// TIA Portal V17 export
// export: Created 2025-05-22T05:59:34.6834771Z, ExportSetting WithDefaults, DisplayName Totally Integrated Automation Portal, DisplayVersion V17 Update 8, DisplayName TIA Portal Openness, DisplayVersion V17 Update 8, DisplayName TIA Portal Version Control Interface, DisplayVersion V17, DisplayName SINAMICS Startdrive Advanced, DisplayVersion V17 SP2, DisplayName SINAMICS Startdrive G110M, G120, G120C, G120D, G120P, G115D, DisplayVersion V17 SP2, DisplayName SINAMICS Startdrive G130, G150, S120, S150, SINAMICS MV, S210, DisplayVersion V17 SP2, DisplayName STEP 7 Professional, DisplayVersion V17 Update 8, DisplayName SINUMERIK ONE STEP 7 Toolbox, DisplayVersion V17 Update 12, DisplayName SINUMERIK ONE PLC Basic Program Plus, DisplayVersion V17 Update 12, DisplayName SINUMERIK 840D sl STEP 7 Toolbox, DisplayVersion V17 Update 12, DisplayName STEP 7 Safety, DisplayVersion V17 Update 6, DisplayName WinCC Advanced, DisplayVersion V17 Update 8
FUNCTION_BLOCK "FB10200_PYROMETERS"   // FB10200, LAD
{ S7_Optimized_Access := 'FALSE' }
AUTHOR : ETXETAR
VERSION : 1.0
// stored: AutoNumber false, IsIECCheckEnabled false, SetENOAutomatically false, UDAEnableTagReadback false
   VAR_INPUT
      OPTIONS_0 : Byte := 2#0000_0000;   // OPTIONS 0
      DEVICE_STATUS_SENSOR_INPUT : Real;   // DEVICE STATUS SENSOR INPUT
      PROCESS_TEMP_SENSOR_INPUT : Real;   // PROCESS TEMPERATURE SENSOR INPUT
      HEAD_TEMP_SENSOR_INPUT : Real;   // HEAD TEMPERATURE SENSOR INPUT
      T1_TEMP_SENSOR_INPUT : Real;   // T1 TEMPERATURE SENSOR INPUT
      T2_TEMP_SENSOR_INPUT : Real;   // T2 TEMPERATURE SENSOR INPUT
      CURRENT_EMISSIVITY_SENSOR_INPUT : Real;   // CURRENT EMISSIVITY SENSOR INPUT
      CURRENT_TRANSMISSION_SENSOR_INPUT : Real;   // CURRENT TRANSMISSION SENSOR INPUT
      STATION_CYCLE_RUNNING : Bool;   // SATION CYCLE RUNNING
   END_VAR
   VAR_OUTPUT
      PROCESS_TEMP_LOW_WARNING : Bool;   // PROCESS TEMPERATURE LOW WARNING
      PROCESS_TEMP_HIGH_WARNING : Bool;   // PROCESS TEMPERATURE HIGH WARNING
      HEAD_TEMP_LOW_WARNING : Bool;   // HEAD TEMPERATURE LOW WARNING
      HEAD_TEMP_HIGH_WARNING : Bool;   // HEAD TEMPERATURE HIGH WARNING
      EMISSIVITY_LOW_WARNING : Bool;   // EMISSIVITY LOW WARNING
      EMISSIVITY_HIGH_WARNING : Bool;   // EMISSIVITY HIGH WARNING
      PROCESS_TEMP_LOW_ALARM : Bool;   // PROCESS TEMPERATURE LOW ALARM
      PROCESS_TEMP_HIGH_ALARM : Bool;   // PROCESS TEMPERATURE HIGH ALARM
      HEAD_TEMP_LOW_ALARM : Bool;   // HEAD TEMPERATURE LOW ALARM
      HEAD_TEMP_HIGH_ALARM : Bool;   // HEAD TEMPERATURE HIGH ALARM
      EMISSIVITY_LOW_ALARM : Bool;   // EMISSIVITY LOW ALARM
      EMISSIVITY_HIGH_ALARM : Bool;   // EMISSIVITY HIGH ALARM
   END_VAR
   VAR DB_SPECIFIC
      ANY_ACTIVE_ALARM : Bool;   // ANY ACTIVE ALARM
      SEOC_ALARMS : Bool;   // STOP END OF CYCLE ALARMS
      RHP_SEOC_ALARMS : Bool;   // RETURN HOME POSITION AND STOP END OF CYCLE ALARMS
      IS_SEOC_ALARMS : Bool;   // INMEDIATE STOP AND STOP END OF CYCLE ALARMS
      UNIT_NUMBER : Int;   // UNIT NUMBER
      PROCESS_TEMP_SETTINGS : Struct
         LOW_WARNING_VALUE : Real;   // LOW WARNING VALUE
         HIGH_WARNING_VALUE : Real;   // HIGH WARNING VALUE
         LOW_ALARM_VALUE : Real;   // LOW ALARM VALUE
         HIGH_ALARM_VALUE : Real;   // HIGH ALARM VALUE
      END_STRUCT;
      HEAD_TEMP_SETTINGS : Struct
         LOW_WARNING_VALUE : Real;   // LOW WARNING VALUE
         HIGH_WARNING_VALUE : Real;   // HIGH WARNING VALUE
         LOW_ALARM_VALUE : Real;   // LOW ALARM VALUE
         HIGH_ALARM_VALUE : Real;   // HIGH ALARM VALUE
      END_STRUCT;
      EMISSIVITY_SETTINGS : Struct
         LOW_WARNING_VALUE : Real;   // LOW WARNING VALUE
         HIGH_WARNING_VALUE : Real;   // HIGH WARNING VALUE
         LOW_ALARM_VALUE : Real;   // LOW ALARM VALUE
         HIGH_ALARM_VALUE : Real;   // HIGH ALARM VALUE
      END_STRUCT;
      TIMERS : Struct
         PROCESS_TEMP_LOW_ALARM_TIMER : TON_TIME;
         PROCESS_TEMP_LOW_WARNING_TIMER : TON_TIME;
         PROCESS_TEMP_HIGH_ALARM_TIMER : TON_TIME;
         PROCESS_TEMP_HIGH_WARNING_TIMER : TON_TIME;
         HEAD_TEMP_LOW_ALARM_TIMER : TON_TIME;
         HEAD_TEMP_LOW_WARNING_TIMER : TON_TIME;
         HEAD_TEMP_HIGH_ALARM_TIMER : TON_TIME;
         HEAD_TEMP_HIGH_WARNING_TIMER : TON_TIME;
         EMISSIVITY_LOW_ALARM_TIMER : TON_TIME;
         EMISSIVITY_LOW_WARNING_TIMER : TON_TIME;
         EMISSIVITY_HIGH_ALARM_TIMER : TON_TIME;
         EMISSIVITY_HIGH_WARNING_TIMER : TON_TIME;
      END_STRUCT;
   END_VAR
   VAR_TEMP
      INPUTS_MASK : Byte;   // INPUT MASK
      O_BYTE_0 : Struct   // OPTIONS BYTE 0
         PROCESS_TEMP_WRNS_ENABLED : Bool;   // PROCESS TEMPERATURE WARNINGS ENABLED
         PROCESS_TEMP_ALARMS_ENABLED : Bool;   // PROCESS TEMPERATURE ALARMS ENABLED
         HEAD_TEMP_WRNS_ENABLED : Bool;   // HEAD TEMPERATURE WARNINGS ENABLED
         HEAD_TEMP_ALARMS_ENABLED : Bool;   // HEAD TEMPERATURE ALARMS ENABLED
         EMISSIVITY_WRNS_ENABLED : Bool;   // EMISSIVITY WARNINGS ENABLED
         EMISSIVITY_ALARMS_ENABLED : Bool;   // EMISSIVITY ALARMS ENABLED
         SPARE_6 : Bool;   // SPARE
         SPARE_7 : Bool;   // SPARE
      END_STRUCT;
      DB_NUMBER : DInt;   // DB NUMBER FOR ALARM AND HELP DECODING
   END_VAR
   VAR_TEMP   // added for the SCL form of the ladder/FBD networks
      _w1 : Bool;
   END_VAR
BEGIN

NETWORK
TITLE = READ INSTANCE DB
      L     DINO;
      +     10#800000;
      T     #DB_NUMBER;


REGION Network 2: OPTIONS
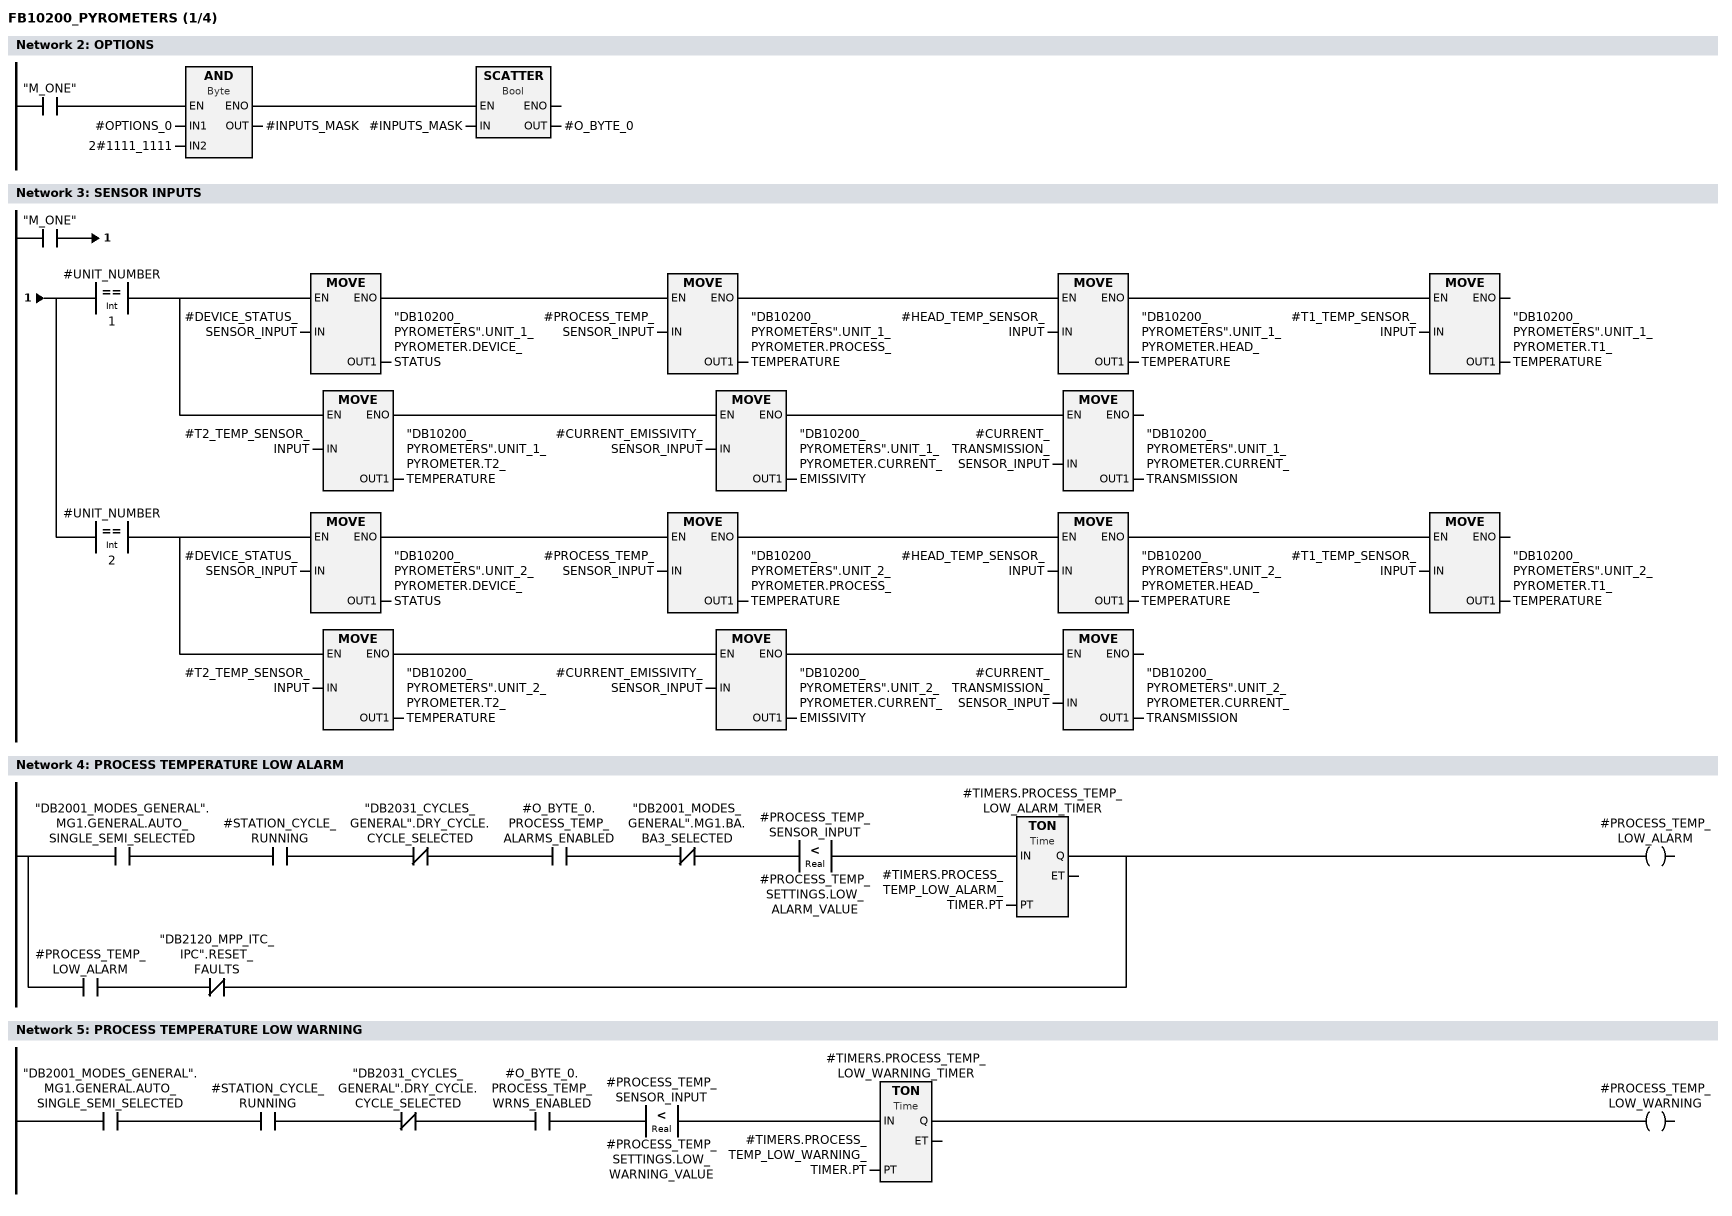
   RUNG wire#powerrail
      Contact( "M_ONE" )
      { S7_Templates := "SrcType := Byte"; S7_GenerateENO := "TRUE" } And(in1 := #OPTIONS_0, in2 := 2#1111_1111, out => #INPUTS_MASK)
      { S7_Templates := "[dest_type := Bool, src_type := Byte]" } SCATTER(IN := #INPUTS_MASK, OUT => #O_BYTE_0)
   END_RUNG
   // the same network as SCL:
   IF "M_ONE" THEN
       #INPUTS_MASK := #OPTIONS_0 AND 2#1111_1111;
       SCATTER(IN := #INPUTS_MASK, OUT => #O_BYTE_0);
   END_IF;
END_REGION

REGION Network 3: SENSOR INPUTS
   RUNG wire#powerrail
      Contact( "M_ONE" )
      wire#w1
      { S7_Templates := "SrcType := Int" } EQ_Contact(in1 := #UNIT_NUMBER, in2 := 1)
      wire#w2
      Move(in := #DEVICE_STATUS_SENSOR_INPUT, out1 => "DB10200_PYROMETERS".UNIT_1_PYROMETER.DEVICE_STATUS)
      Move(in := #PROCESS_TEMP_SENSOR_INPUT, out1 => "DB10200_PYROMETERS".UNIT_1_PYROMETER.PROCESS_TEMPERATURE)
      Move(in := #HEAD_TEMP_SENSOR_INPUT, out1 => "DB10200_PYROMETERS".UNIT_1_PYROMETER.HEAD_TEMPERATURE)
      Move(in := #T1_TEMP_SENSOR_INPUT, out1 => "DB10200_PYROMETERS".UNIT_1_PYROMETER.T1_TEMPERATURE)
   END_RUNG
   RUNG wire#w2
      Move(in := #T2_TEMP_SENSOR_INPUT, out1 => "DB10200_PYROMETERS".UNIT_1_PYROMETER.T2_TEMPERATURE)
      Move(in := #CURRENT_EMISSIVITY_SENSOR_INPUT, out1 => "DB10200_PYROMETERS".UNIT_1_PYROMETER.CURRENT_EMISSIVITY)
      Move(in := #CURRENT_TRANSMISSION_SENSOR_INPUT, out1 => "DB10200_PYROMETERS".UNIT_1_PYROMETER.CURRENT_TRANSMISSION)
   END_RUNG
   RUNG wire#w1
      { S7_Templates := "SrcType := Int" } EQ_Contact(in1 := #UNIT_NUMBER, in2 := 2)
      wire#w3
      Move(in := #DEVICE_STATUS_SENSOR_INPUT, out1 => "DB10200_PYROMETERS".UNIT_2_PYROMETER.DEVICE_STATUS)
      Move(in := #PROCESS_TEMP_SENSOR_INPUT, out1 => "DB10200_PYROMETERS".UNIT_2_PYROMETER.PROCESS_TEMPERATURE)
      Move(in := #HEAD_TEMP_SENSOR_INPUT, out1 => "DB10200_PYROMETERS".UNIT_2_PYROMETER.HEAD_TEMPERATURE)
      Move(in := #T1_TEMP_SENSOR_INPUT, out1 => "DB10200_PYROMETERS".UNIT_2_PYROMETER.T1_TEMPERATURE)
   END_RUNG
   RUNG wire#w3
      Move(in := #T2_TEMP_SENSOR_INPUT, out1 => "DB10200_PYROMETERS".UNIT_2_PYROMETER.T2_TEMPERATURE)
      Move(in := #CURRENT_EMISSIVITY_SENSOR_INPUT, out1 => "DB10200_PYROMETERS".UNIT_2_PYROMETER.CURRENT_EMISSIVITY)
      Move(in := #CURRENT_TRANSMISSION_SENSOR_INPUT, out1 => "DB10200_PYROMETERS".UNIT_2_PYROMETER.CURRENT_TRANSMISSION)
   END_RUNG
   // the same network as SCL:
   IF "M_ONE" AND (#UNIT_NUMBER = 1) THEN
       "DB10200_PYROMETERS".UNIT_1_PYROMETER.DEVICE_STATUS := #DEVICE_STATUS_SENSOR_INPUT;
       "DB10200_PYROMETERS".UNIT_1_PYROMETER.PROCESS_TEMPERATURE := #PROCESS_TEMP_SENSOR_INPUT;
       "DB10200_PYROMETERS".UNIT_1_PYROMETER.HEAD_TEMPERATURE := #HEAD_TEMP_SENSOR_INPUT;
       "DB10200_PYROMETERS".UNIT_1_PYROMETER.T1_TEMPERATURE := #T1_TEMP_SENSOR_INPUT;
       "DB10200_PYROMETERS".UNIT_1_PYROMETER.T2_TEMPERATURE := #T2_TEMP_SENSOR_INPUT;
       "DB10200_PYROMETERS".UNIT_1_PYROMETER.CURRENT_EMISSIVITY := #CURRENT_EMISSIVITY_SENSOR_INPUT;
       "DB10200_PYROMETERS".UNIT_1_PYROMETER.CURRENT_TRANSMISSION := #CURRENT_TRANSMISSION_SENSOR_INPUT;
   END_IF;
   IF "M_ONE" AND (#UNIT_NUMBER = 2) THEN
       "DB10200_PYROMETERS".UNIT_2_PYROMETER.DEVICE_STATUS := #DEVICE_STATUS_SENSOR_INPUT;
       "DB10200_PYROMETERS".UNIT_2_PYROMETER.PROCESS_TEMPERATURE := #PROCESS_TEMP_SENSOR_INPUT;
       "DB10200_PYROMETERS".UNIT_2_PYROMETER.HEAD_TEMPERATURE := #HEAD_TEMP_SENSOR_INPUT;
       "DB10200_PYROMETERS".UNIT_2_PYROMETER.T1_TEMPERATURE := #T1_TEMP_SENSOR_INPUT;
       "DB10200_PYROMETERS".UNIT_2_PYROMETER.T2_TEMPERATURE := #T2_TEMP_SENSOR_INPUT;
       "DB10200_PYROMETERS".UNIT_2_PYROMETER.CURRENT_EMISSIVITY := #CURRENT_EMISSIVITY_SENSOR_INPUT;
       "DB10200_PYROMETERS".UNIT_2_PYROMETER.CURRENT_TRANSMISSION := #CURRENT_TRANSMISSION_SENSOR_INPUT;
   END_IF;
END_REGION

REGION Network 4: PROCESS TEMPERATURE LOW ALARM
   RUNG wire#powerrail
      Contact( "DB2001_MODES_GENERAL".MG1.GENERAL.AUTO_SINGLE_SEMI_SELECTED )
      Contact( #STATION_CYCLE_RUNNING )
      I_Contact( "DB2031_CYCLES_GENERAL".DRY_CYCLE.CYCLE_SELECTED )
      Contact( #O_BYTE_0.PROCESS_TEMP_ALARMS_ENABLED )
      I_Contact( "DB2001_MODES_GENERAL".MG1.BA.BA3_SELECTED )
      { S7_Templates := "SrcType := Real" } LT_Contact(in1 := #PROCESS_TEMP_SENSOR_INPUT, in2 := #PROCESS_TEMP_SETTINGS.LOW_ALARM_VALUE)
      { S7_Templates := "time_type := Time" } #TIMERS.PROCESS_TEMP_LOW_ALARM_TIMER.TON(pt := #TIMERS.PROCESS_TEMP_LOW_ALARM_TIMER.PT, et =>)
      wire#w1
      Coil( #PROCESS_TEMP_LOW_ALARM )
   END_RUNG
   RUNG wire#powerrail
      Contact( #PROCESS_TEMP_LOW_ALARM )
      I_Contact( "DB2120_MPP_ITC_IPC".RESET_FAULTS )
   END_RUNG wire#w1
   // the same network as SCL:
   #TIMERS.PROCESS_TEMP_LOW_ALARM_TIMER.TON(IN := "DB2001_MODES_GENERAL".MG1.GENERAL.AUTO_SINGLE_SEMI_SELECTED AND #STATION_CYCLE_RUNNING AND NOT "DB2031_CYCLES_GENERAL".DRY_CYCLE.CYCLE_SELECTED AND #O_BYTE_0.PROCESS_TEMP_ALARMS_ENABLED AND NOT "DB2001_MODES_GENERAL".MG1.BA.BA3_SELECTED AND (#PROCESS_TEMP_SENSOR_INPUT < #PROCESS_TEMP_SETTINGS.LOW_ALARM_VALUE),
                           PT := #TIMERS.PROCESS_TEMP_LOW_ALARM_TIMER.PT);
   #PROCESS_TEMP_LOW_ALARM := #TIMERS.PROCESS_TEMP_LOW_ALARM_TIMER.Q OR (#PROCESS_TEMP_LOW_ALARM AND NOT "DB2120_MPP_ITC_IPC".RESET_FAULTS);
END_REGION

REGION Network 5: PROCESS TEMPERATURE LOW WARNING
   RUNG wire#powerrail
      Contact( "DB2001_MODES_GENERAL".MG1.GENERAL.AUTO_SINGLE_SEMI_SELECTED )
      Contact( #STATION_CYCLE_RUNNING )
      I_Contact( "DB2031_CYCLES_GENERAL".DRY_CYCLE.CYCLE_SELECTED )
      Contact( #O_BYTE_0.PROCESS_TEMP_WRNS_ENABLED )
      { S7_Templates := "SrcType := Real" } LT_Contact(in1 := #PROCESS_TEMP_SENSOR_INPUT, in2 := #PROCESS_TEMP_SETTINGS.LOW_WARNING_VALUE)
      { S7_Templates := "time_type := Time" } #TIMERS.PROCESS_TEMP_LOW_WARNING_TIMER.TON(pt := #TIMERS.PROCESS_TEMP_LOW_WARNING_TIMER.PT, et =>)
      Coil( #PROCESS_TEMP_LOW_WARNING )
   END_RUNG
   // the same network as SCL:
   #TIMERS.PROCESS_TEMP_LOW_WARNING_TIMER.TON(IN := "DB2001_MODES_GENERAL".MG1.GENERAL.AUTO_SINGLE_SEMI_SELECTED AND #STATION_CYCLE_RUNNING AND NOT "DB2031_CYCLES_GENERAL".DRY_CYCLE.CYCLE_SELECTED AND #O_BYTE_0.PROCESS_TEMP_WRNS_ENABLED AND (#PROCESS_TEMP_SENSOR_INPUT < #PROCESS_TEMP_SETTINGS.LOW_WARNING_VALUE),
                           PT := #TIMERS.PROCESS_TEMP_LOW_WARNING_TIMER.PT);
   #PROCESS_TEMP_LOW_WARNING := #TIMERS.PROCESS_TEMP_LOW_WARNING_TIMER.Q;
END_REGION

REGION Network 6: PROCESS TEMPERATURE HIGH ALARM
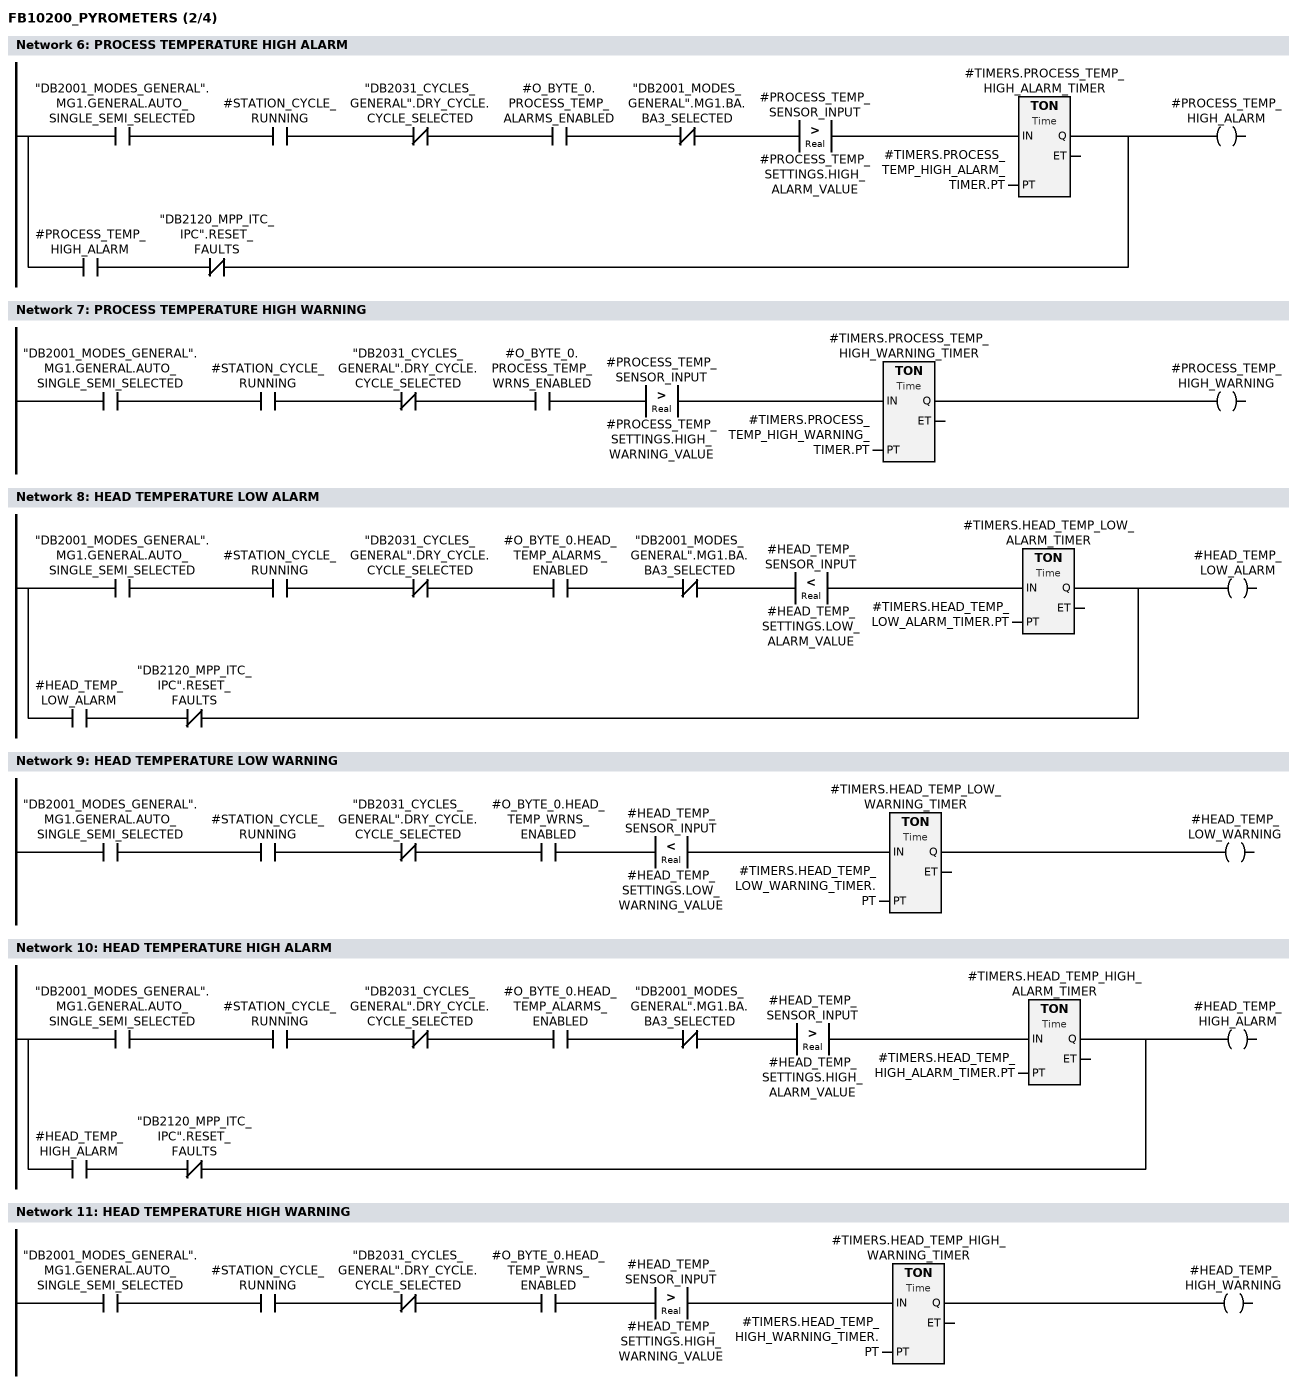
   RUNG wire#powerrail
      Contact( "DB2001_MODES_GENERAL".MG1.GENERAL.AUTO_SINGLE_SEMI_SELECTED )
      Contact( #STATION_CYCLE_RUNNING )
      I_Contact( "DB2031_CYCLES_GENERAL".DRY_CYCLE.CYCLE_SELECTED )
      Contact( #O_BYTE_0.PROCESS_TEMP_ALARMS_ENABLED )
      I_Contact( "DB2001_MODES_GENERAL".MG1.BA.BA3_SELECTED )
      { S7_Templates := "SrcType := Real" } GT_Contact(in1 := #PROCESS_TEMP_SENSOR_INPUT, in2 := #PROCESS_TEMP_SETTINGS.HIGH_ALARM_VALUE)
      { S7_Templates := "time_type := Time" } #TIMERS.PROCESS_TEMP_HIGH_ALARM_TIMER.TON(pt := #TIMERS.PROCESS_TEMP_HIGH_ALARM_TIMER.PT, et =>)
      wire#w1
      Coil( #PROCESS_TEMP_HIGH_ALARM )
   END_RUNG
   RUNG wire#powerrail
      Contact( #PROCESS_TEMP_HIGH_ALARM )
      I_Contact( "DB2120_MPP_ITC_IPC".RESET_FAULTS )
   END_RUNG wire#w1
   // the same network as SCL:
   #TIMERS.PROCESS_TEMP_HIGH_ALARM_TIMER.TON(IN := "DB2001_MODES_GENERAL".MG1.GENERAL.AUTO_SINGLE_SEMI_SELECTED AND #STATION_CYCLE_RUNNING AND NOT "DB2031_CYCLES_GENERAL".DRY_CYCLE.CYCLE_SELECTED AND #O_BYTE_0.PROCESS_TEMP_ALARMS_ENABLED AND NOT "DB2001_MODES_GENERAL".MG1.BA.BA3_SELECTED AND (#PROCESS_TEMP_SENSOR_INPUT > #PROCESS_TEMP_SETTINGS.HIGH_ALARM_VALUE),
                           PT := #TIMERS.PROCESS_TEMP_HIGH_ALARM_TIMER.PT);
   #PROCESS_TEMP_HIGH_ALARM := #TIMERS.PROCESS_TEMP_HIGH_ALARM_TIMER.Q OR (#PROCESS_TEMP_HIGH_ALARM AND NOT "DB2120_MPP_ITC_IPC".RESET_FAULTS);
END_REGION

REGION Network 7: PROCESS TEMPERATURE HIGH WARNING
   RUNG wire#powerrail
      Contact( "DB2001_MODES_GENERAL".MG1.GENERAL.AUTO_SINGLE_SEMI_SELECTED )
      Contact( #STATION_CYCLE_RUNNING )
      I_Contact( "DB2031_CYCLES_GENERAL".DRY_CYCLE.CYCLE_SELECTED )
      Contact( #O_BYTE_0.PROCESS_TEMP_WRNS_ENABLED )
      { S7_Templates := "SrcType := Real" } GT_Contact(in1 := #PROCESS_TEMP_SENSOR_INPUT, in2 := #PROCESS_TEMP_SETTINGS.HIGH_WARNING_VALUE)
      { S7_Templates := "time_type := Time" } #TIMERS.PROCESS_TEMP_HIGH_WARNING_TIMER.TON(pt := #TIMERS.PROCESS_TEMP_HIGH_WARNING_TIMER.PT, et =>)
      Coil( #PROCESS_TEMP_HIGH_WARNING )
   END_RUNG
   // the same network as SCL:
   #TIMERS.PROCESS_TEMP_HIGH_WARNING_TIMER.TON(IN := "DB2001_MODES_GENERAL".MG1.GENERAL.AUTO_SINGLE_SEMI_SELECTED AND #STATION_CYCLE_RUNNING AND NOT "DB2031_CYCLES_GENERAL".DRY_CYCLE.CYCLE_SELECTED AND #O_BYTE_0.PROCESS_TEMP_WRNS_ENABLED AND (#PROCESS_TEMP_SENSOR_INPUT > #PROCESS_TEMP_SETTINGS.HIGH_WARNING_VALUE),
                           PT := #TIMERS.PROCESS_TEMP_HIGH_WARNING_TIMER.PT);
   #PROCESS_TEMP_HIGH_WARNING := #TIMERS.PROCESS_TEMP_HIGH_WARNING_TIMER.Q;
END_REGION

REGION Network 8: HEAD TEMPERATURE LOW ALARM
   RUNG wire#powerrail
      Contact( "DB2001_MODES_GENERAL".MG1.GENERAL.AUTO_SINGLE_SEMI_SELECTED )
      Contact( #STATION_CYCLE_RUNNING )
      I_Contact( "DB2031_CYCLES_GENERAL".DRY_CYCLE.CYCLE_SELECTED )
      Contact( #O_BYTE_0.HEAD_TEMP_ALARMS_ENABLED )
      I_Contact( "DB2001_MODES_GENERAL".MG1.BA.BA3_SELECTED )
      { S7_Templates := "SrcType := Real" } LT_Contact(in1 := #HEAD_TEMP_SENSOR_INPUT, in2 := #HEAD_TEMP_SETTINGS.LOW_ALARM_VALUE)
      { S7_Templates := "time_type := Time" } #TIMERS.HEAD_TEMP_LOW_ALARM_TIMER.TON(pt := #TIMERS.HEAD_TEMP_LOW_ALARM_TIMER.PT, et =>)
      wire#w1
      Coil( #HEAD_TEMP_LOW_ALARM )
   END_RUNG
   RUNG wire#powerrail
      Contact( #HEAD_TEMP_LOW_ALARM )
      I_Contact( "DB2120_MPP_ITC_IPC".RESET_FAULTS )
   END_RUNG wire#w1
   // the same network as SCL:
   #TIMERS.HEAD_TEMP_LOW_ALARM_TIMER.TON(IN := "DB2001_MODES_GENERAL".MG1.GENERAL.AUTO_SINGLE_SEMI_SELECTED AND #STATION_CYCLE_RUNNING AND NOT "DB2031_CYCLES_GENERAL".DRY_CYCLE.CYCLE_SELECTED AND #O_BYTE_0.HEAD_TEMP_ALARMS_ENABLED AND NOT "DB2001_MODES_GENERAL".MG1.BA.BA3_SELECTED AND (#HEAD_TEMP_SENSOR_INPUT < #HEAD_TEMP_SETTINGS.LOW_ALARM_VALUE),
                           PT := #TIMERS.HEAD_TEMP_LOW_ALARM_TIMER.PT);
   #HEAD_TEMP_LOW_ALARM := #TIMERS.HEAD_TEMP_LOW_ALARM_TIMER.Q OR (#HEAD_TEMP_LOW_ALARM AND NOT "DB2120_MPP_ITC_IPC".RESET_FAULTS);
END_REGION

REGION Network 9: HEAD TEMPERATURE LOW WARNING
   RUNG wire#powerrail
      Contact( "DB2001_MODES_GENERAL".MG1.GENERAL.AUTO_SINGLE_SEMI_SELECTED )
      Contact( #STATION_CYCLE_RUNNING )
      I_Contact( "DB2031_CYCLES_GENERAL".DRY_CYCLE.CYCLE_SELECTED )
      Contact( #O_BYTE_0.HEAD_TEMP_WRNS_ENABLED )
      { S7_Templates := "SrcType := Real" } LT_Contact(in1 := #HEAD_TEMP_SENSOR_INPUT, in2 := #HEAD_TEMP_SETTINGS.LOW_WARNING_VALUE)
      { S7_Templates := "time_type := Time" } #TIMERS.HEAD_TEMP_LOW_WARNING_TIMER.TON(pt := #TIMERS.HEAD_TEMP_LOW_WARNING_TIMER.PT, et =>)
      Coil( #HEAD_TEMP_LOW_WARNING )
   END_RUNG
   // the same network as SCL:
   #TIMERS.HEAD_TEMP_LOW_WARNING_TIMER.TON(IN := "DB2001_MODES_GENERAL".MG1.GENERAL.AUTO_SINGLE_SEMI_SELECTED AND #STATION_CYCLE_RUNNING AND NOT "DB2031_CYCLES_GENERAL".DRY_CYCLE.CYCLE_SELECTED AND #O_BYTE_0.HEAD_TEMP_WRNS_ENABLED AND (#HEAD_TEMP_SENSOR_INPUT < #HEAD_TEMP_SETTINGS.LOW_WARNING_VALUE),
                           PT := #TIMERS.HEAD_TEMP_LOW_WARNING_TIMER.PT);
   #HEAD_TEMP_LOW_WARNING := #TIMERS.HEAD_TEMP_LOW_WARNING_TIMER.Q;
END_REGION

REGION Network 10: HEAD TEMPERATURE HIGH ALARM
   RUNG wire#powerrail
      Contact( "DB2001_MODES_GENERAL".MG1.GENERAL.AUTO_SINGLE_SEMI_SELECTED )
      Contact( #STATION_CYCLE_RUNNING )
      I_Contact( "DB2031_CYCLES_GENERAL".DRY_CYCLE.CYCLE_SELECTED )
      Contact( #O_BYTE_0.HEAD_TEMP_ALARMS_ENABLED )
      I_Contact( "DB2001_MODES_GENERAL".MG1.BA.BA3_SELECTED )
      { S7_Templates := "SrcType := Real" } GT_Contact(in1 := #HEAD_TEMP_SENSOR_INPUT, in2 := #HEAD_TEMP_SETTINGS.HIGH_ALARM_VALUE)
      { S7_Templates := "time_type := Time" } #TIMERS.HEAD_TEMP_HIGH_ALARM_TIMER.TON(pt := #TIMERS.HEAD_TEMP_HIGH_ALARM_TIMER.PT, et =>)
      wire#w1
      Coil( #HEAD_TEMP_HIGH_ALARM )
   END_RUNG
   RUNG wire#powerrail
      Contact( #HEAD_TEMP_HIGH_ALARM )
      I_Contact( "DB2120_MPP_ITC_IPC".RESET_FAULTS )
   END_RUNG wire#w1
   // the same network as SCL:
   #TIMERS.HEAD_TEMP_HIGH_ALARM_TIMER.TON(IN := "DB2001_MODES_GENERAL".MG1.GENERAL.AUTO_SINGLE_SEMI_SELECTED AND #STATION_CYCLE_RUNNING AND NOT "DB2031_CYCLES_GENERAL".DRY_CYCLE.CYCLE_SELECTED AND #O_BYTE_0.HEAD_TEMP_ALARMS_ENABLED AND NOT "DB2001_MODES_GENERAL".MG1.BA.BA3_SELECTED AND (#HEAD_TEMP_SENSOR_INPUT > #HEAD_TEMP_SETTINGS.HIGH_ALARM_VALUE),
                           PT := #TIMERS.HEAD_TEMP_HIGH_ALARM_TIMER.PT);
   #HEAD_TEMP_HIGH_ALARM := #TIMERS.HEAD_TEMP_HIGH_ALARM_TIMER.Q OR (#HEAD_TEMP_HIGH_ALARM AND NOT "DB2120_MPP_ITC_IPC".RESET_FAULTS);
END_REGION

REGION Network 11: HEAD TEMPERATURE HIGH WARNING
   RUNG wire#powerrail
      Contact( "DB2001_MODES_GENERAL".MG1.GENERAL.AUTO_SINGLE_SEMI_SELECTED )
      Contact( #STATION_CYCLE_RUNNING )
      I_Contact( "DB2031_CYCLES_GENERAL".DRY_CYCLE.CYCLE_SELECTED )
      Contact( #O_BYTE_0.HEAD_TEMP_WRNS_ENABLED )
      { S7_Templates := "SrcType := Real" } GT_Contact(in1 := #HEAD_TEMP_SENSOR_INPUT, in2 := #HEAD_TEMP_SETTINGS.HIGH_WARNING_VALUE)
      { S7_Templates := "time_type := Time" } #TIMERS.HEAD_TEMP_HIGH_WARNING_TIMER.TON(pt := #TIMERS.HEAD_TEMP_HIGH_WARNING_TIMER.PT, et =>)
      Coil( #HEAD_TEMP_HIGH_WARNING )
   END_RUNG
   // the same network as SCL:
   #TIMERS.HEAD_TEMP_HIGH_WARNING_TIMER.TON(IN := "DB2001_MODES_GENERAL".MG1.GENERAL.AUTO_SINGLE_SEMI_SELECTED AND #STATION_CYCLE_RUNNING AND NOT "DB2031_CYCLES_GENERAL".DRY_CYCLE.CYCLE_SELECTED AND #O_BYTE_0.HEAD_TEMP_WRNS_ENABLED AND (#HEAD_TEMP_SENSOR_INPUT > #HEAD_TEMP_SETTINGS.HIGH_WARNING_VALUE),
                           PT := #TIMERS.HEAD_TEMP_HIGH_WARNING_TIMER.PT);
   #HEAD_TEMP_HIGH_WARNING := #TIMERS.HEAD_TEMP_HIGH_WARNING_TIMER.Q;
END_REGION

REGION Network 12: EMISSIVITY LOW ALARM
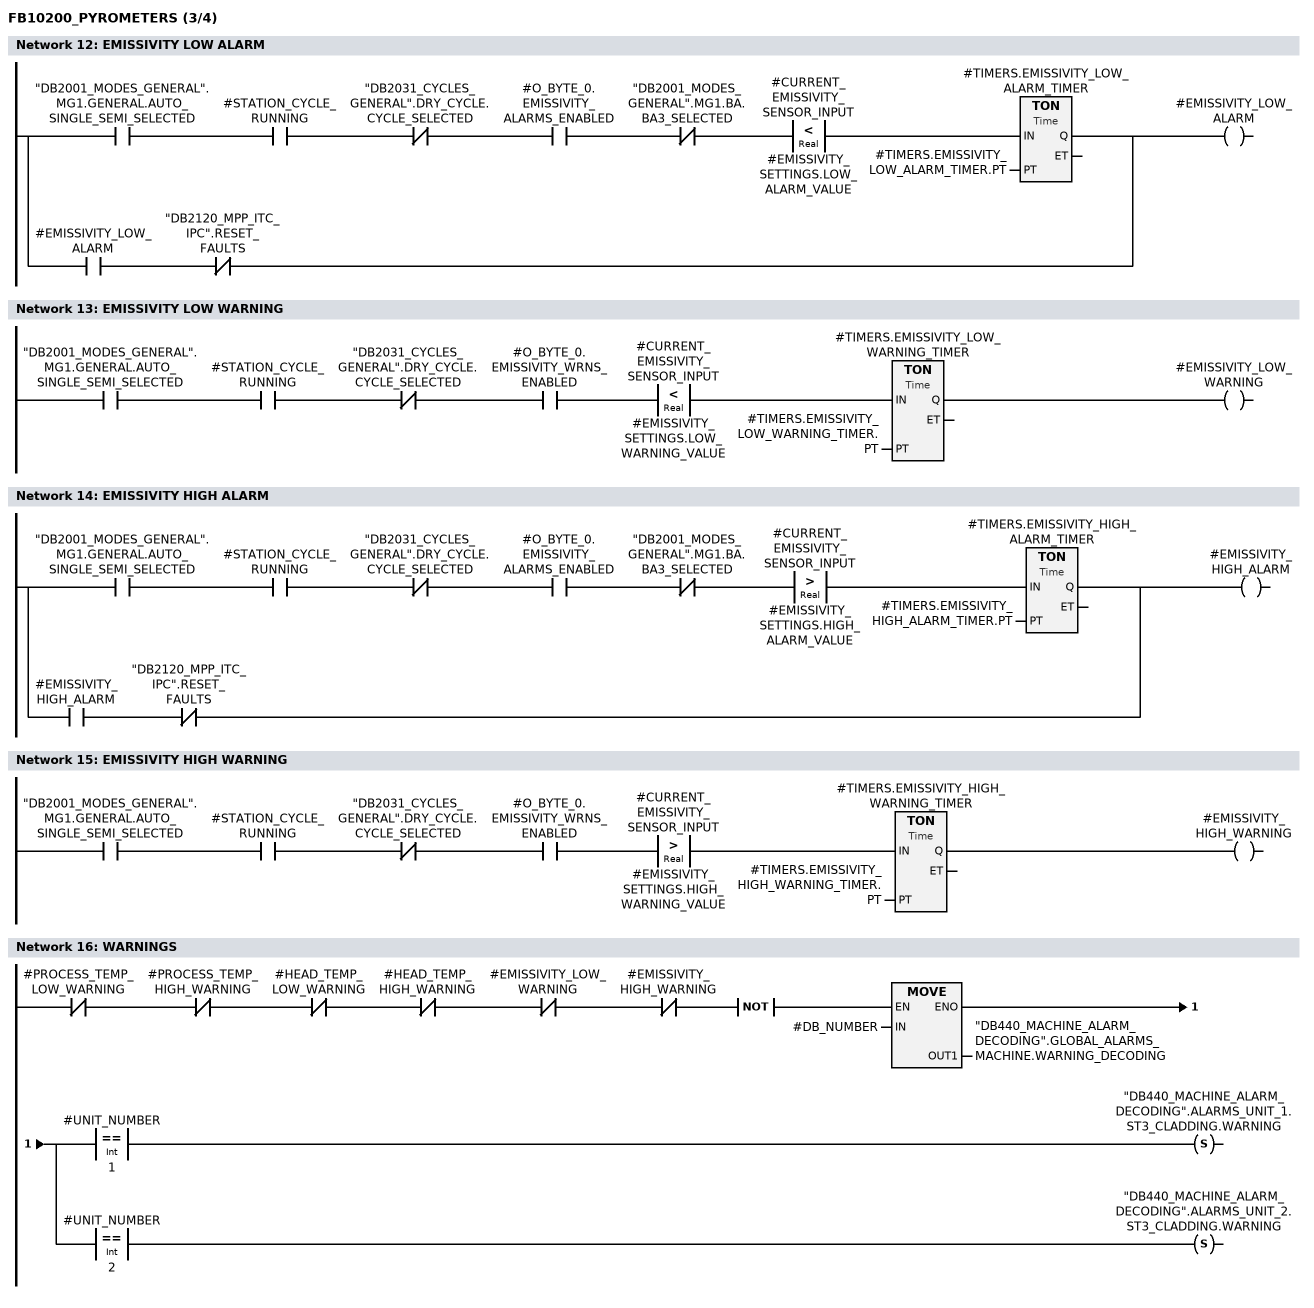
   RUNG wire#powerrail
      Contact( "DB2001_MODES_GENERAL".MG1.GENERAL.AUTO_SINGLE_SEMI_SELECTED )
      Contact( #STATION_CYCLE_RUNNING )
      I_Contact( "DB2031_CYCLES_GENERAL".DRY_CYCLE.CYCLE_SELECTED )
      Contact( #O_BYTE_0.EMISSIVITY_ALARMS_ENABLED )
      I_Contact( "DB2001_MODES_GENERAL".MG1.BA.BA3_SELECTED )
      { S7_Templates := "SrcType := Real" } LT_Contact(in1 := #CURRENT_EMISSIVITY_SENSOR_INPUT, in2 := #EMISSIVITY_SETTINGS.LOW_ALARM_VALUE)
      { S7_Templates := "time_type := Time" } #TIMERS.EMISSIVITY_LOW_ALARM_TIMER.TON(pt := #TIMERS.EMISSIVITY_LOW_ALARM_TIMER.PT, et =>)
      wire#w1
      Coil( #EMISSIVITY_LOW_ALARM )
   END_RUNG
   RUNG wire#powerrail
      Contact( #EMISSIVITY_LOW_ALARM )
      I_Contact( "DB2120_MPP_ITC_IPC".RESET_FAULTS )
   END_RUNG wire#w1
   // the same network as SCL:
   #TIMERS.EMISSIVITY_LOW_ALARM_TIMER.TON(IN := "DB2001_MODES_GENERAL".MG1.GENERAL.AUTO_SINGLE_SEMI_SELECTED AND #STATION_CYCLE_RUNNING AND NOT "DB2031_CYCLES_GENERAL".DRY_CYCLE.CYCLE_SELECTED AND #O_BYTE_0.EMISSIVITY_ALARMS_ENABLED AND NOT "DB2001_MODES_GENERAL".MG1.BA.BA3_SELECTED AND (#CURRENT_EMISSIVITY_SENSOR_INPUT < #EMISSIVITY_SETTINGS.LOW_ALARM_VALUE),
                           PT := #TIMERS.EMISSIVITY_LOW_ALARM_TIMER.PT);
   #EMISSIVITY_LOW_ALARM := #TIMERS.EMISSIVITY_LOW_ALARM_TIMER.Q OR (#EMISSIVITY_LOW_ALARM AND NOT "DB2120_MPP_ITC_IPC".RESET_FAULTS);
END_REGION

REGION Network 13: EMISSIVITY LOW WARNING
   RUNG wire#powerrail
      Contact( "DB2001_MODES_GENERAL".MG1.GENERAL.AUTO_SINGLE_SEMI_SELECTED )
      Contact( #STATION_CYCLE_RUNNING )
      I_Contact( "DB2031_CYCLES_GENERAL".DRY_CYCLE.CYCLE_SELECTED )
      Contact( #O_BYTE_0.EMISSIVITY_WRNS_ENABLED )
      { S7_Templates := "SrcType := Real" } LT_Contact(in1 := #CURRENT_EMISSIVITY_SENSOR_INPUT, in2 := #EMISSIVITY_SETTINGS.LOW_WARNING_VALUE)
      { S7_Templates := "time_type := Time" } #TIMERS.EMISSIVITY_LOW_WARNING_TIMER.TON(pt := #TIMERS.EMISSIVITY_LOW_WARNING_TIMER.PT, et =>)
      Coil( #EMISSIVITY_LOW_WARNING )
   END_RUNG
   // the same network as SCL:
   #TIMERS.EMISSIVITY_LOW_WARNING_TIMER.TON(IN := "DB2001_MODES_GENERAL".MG1.GENERAL.AUTO_SINGLE_SEMI_SELECTED AND #STATION_CYCLE_RUNNING AND NOT "DB2031_CYCLES_GENERAL".DRY_CYCLE.CYCLE_SELECTED AND #O_BYTE_0.EMISSIVITY_WRNS_ENABLED AND (#CURRENT_EMISSIVITY_SENSOR_INPUT < #EMISSIVITY_SETTINGS.LOW_WARNING_VALUE),
                           PT := #TIMERS.EMISSIVITY_LOW_WARNING_TIMER.PT);
   #EMISSIVITY_LOW_WARNING := #TIMERS.EMISSIVITY_LOW_WARNING_TIMER.Q;
END_REGION

REGION Network 14: EMISSIVITY HIGH ALARM
   RUNG wire#powerrail
      Contact( "DB2001_MODES_GENERAL".MG1.GENERAL.AUTO_SINGLE_SEMI_SELECTED )
      Contact( #STATION_CYCLE_RUNNING )
      I_Contact( "DB2031_CYCLES_GENERAL".DRY_CYCLE.CYCLE_SELECTED )
      Contact( #O_BYTE_0.EMISSIVITY_ALARMS_ENABLED )
      I_Contact( "DB2001_MODES_GENERAL".MG1.BA.BA3_SELECTED )
      { S7_Templates := "SrcType := Real" } GT_Contact(in1 := #CURRENT_EMISSIVITY_SENSOR_INPUT, in2 := #EMISSIVITY_SETTINGS.HIGH_ALARM_VALUE)
      { S7_Templates := "time_type := Time" } #TIMERS.EMISSIVITY_HIGH_ALARM_TIMER.TON(pt := #TIMERS.EMISSIVITY_HIGH_ALARM_TIMER.PT, et =>)
      wire#w1
      Coil( #EMISSIVITY_HIGH_ALARM )
   END_RUNG
   RUNG wire#powerrail
      Contact( #EMISSIVITY_HIGH_ALARM )
      I_Contact( "DB2120_MPP_ITC_IPC".RESET_FAULTS )
   END_RUNG wire#w1
   // the same network as SCL:
   #TIMERS.EMISSIVITY_HIGH_ALARM_TIMER.TON(IN := "DB2001_MODES_GENERAL".MG1.GENERAL.AUTO_SINGLE_SEMI_SELECTED AND #STATION_CYCLE_RUNNING AND NOT "DB2031_CYCLES_GENERAL".DRY_CYCLE.CYCLE_SELECTED AND #O_BYTE_0.EMISSIVITY_ALARMS_ENABLED AND NOT "DB2001_MODES_GENERAL".MG1.BA.BA3_SELECTED AND (#CURRENT_EMISSIVITY_SENSOR_INPUT > #EMISSIVITY_SETTINGS.HIGH_ALARM_VALUE),
                           PT := #TIMERS.EMISSIVITY_HIGH_ALARM_TIMER.PT);
   #EMISSIVITY_HIGH_ALARM := #TIMERS.EMISSIVITY_HIGH_ALARM_TIMER.Q OR (#EMISSIVITY_HIGH_ALARM AND NOT "DB2120_MPP_ITC_IPC".RESET_FAULTS);
END_REGION

REGION Network 15: EMISSIVITY HIGH WARNING
   RUNG wire#powerrail
      Contact( "DB2001_MODES_GENERAL".MG1.GENERAL.AUTO_SINGLE_SEMI_SELECTED )
      Contact( #STATION_CYCLE_RUNNING )
      I_Contact( "DB2031_CYCLES_GENERAL".DRY_CYCLE.CYCLE_SELECTED )
      Contact( #O_BYTE_0.EMISSIVITY_WRNS_ENABLED )
      { S7_Templates := "SrcType := Real" } GT_Contact(in1 := #CURRENT_EMISSIVITY_SENSOR_INPUT, in2 := #EMISSIVITY_SETTINGS.HIGH_WARNING_VALUE)
      { S7_Templates := "time_type := Time" } #TIMERS.EMISSIVITY_HIGH_WARNING_TIMER.TON(pt := #TIMERS.EMISSIVITY_HIGH_WARNING_TIMER.PT, et =>)
      Coil( #EMISSIVITY_HIGH_WARNING )
   END_RUNG
   // the same network as SCL:
   #TIMERS.EMISSIVITY_HIGH_WARNING_TIMER.TON(IN := "DB2001_MODES_GENERAL".MG1.GENERAL.AUTO_SINGLE_SEMI_SELECTED AND #STATION_CYCLE_RUNNING AND NOT "DB2031_CYCLES_GENERAL".DRY_CYCLE.CYCLE_SELECTED AND #O_BYTE_0.EMISSIVITY_WRNS_ENABLED AND (#CURRENT_EMISSIVITY_SENSOR_INPUT > #EMISSIVITY_SETTINGS.HIGH_WARNING_VALUE),
                           PT := #TIMERS.EMISSIVITY_HIGH_WARNING_TIMER.PT);
   #EMISSIVITY_HIGH_WARNING := #TIMERS.EMISSIVITY_HIGH_WARNING_TIMER.Q;
END_REGION

REGION Network 16: WARNINGS
   RUNG wire#powerrail
      I_Contact( #PROCESS_TEMP_LOW_WARNING )
      I_Contact( #PROCESS_TEMP_HIGH_WARNING )
      I_Contact( #HEAD_TEMP_LOW_WARNING )
      I_Contact( #HEAD_TEMP_HIGH_WARNING )
      I_Contact( #EMISSIVITY_LOW_WARNING )
      I_Contact( #EMISSIVITY_HIGH_WARNING )
      Not()
      Move(in := #DB_NUMBER, out1 => "DB440_MACHINE_ALARM_DECODING".GLOBAL_ALARMS_MACHINE.WARNING_DECODING)
      wire#w1
      { S7_Templates := "SrcType := Int" } EQ_Contact(in1 := #UNIT_NUMBER, in2 := 1)
      S_Coil( "DB440_MACHINE_ALARM_DECODING".ALARMS_UNIT_1.ST3_CLADDING.WARNING )
   END_RUNG
   RUNG wire#w1
      { S7_Templates := "SrcType := Int" } EQ_Contact(in1 := #UNIT_NUMBER, in2 := 2)
      S_Coil( "DB440_MACHINE_ALARM_DECODING".ALARMS_UNIT_2.ST3_CLADDING.WARNING )
   END_RUNG
   // the same network as SCL:
   #_w1 := NOT (NOT #PROCESS_TEMP_LOW_WARNING AND NOT #PROCESS_TEMP_HIGH_WARNING AND NOT #HEAD_TEMP_LOW_WARNING AND NOT #HEAD_TEMP_HIGH_WARNING AND NOT #EMISSIVITY_LOW_WARNING AND NOT #EMISSIVITY_HIGH_WARNING);
   IF #_w1 THEN "DB440_MACHINE_ALARM_DECODING".GLOBAL_ALARMS_MACHINE.WARNING_DECODING := #DB_NUMBER; END_IF;
   IF #_w1 AND (#UNIT_NUMBER = 1) THEN
       "DB440_MACHINE_ALARM_DECODING".ALARMS_UNIT_1.ST3_CLADDING.WARNING := TRUE;
   END_IF;
   IF #_w1 AND (#UNIT_NUMBER = 2) THEN
       "DB440_MACHINE_ALARM_DECODING".ALARMS_UNIT_2.ST3_CLADDING.WARNING := TRUE;
   END_IF;
END_REGION

REGION Network 17: STOP END OF CYCLE ALARMS
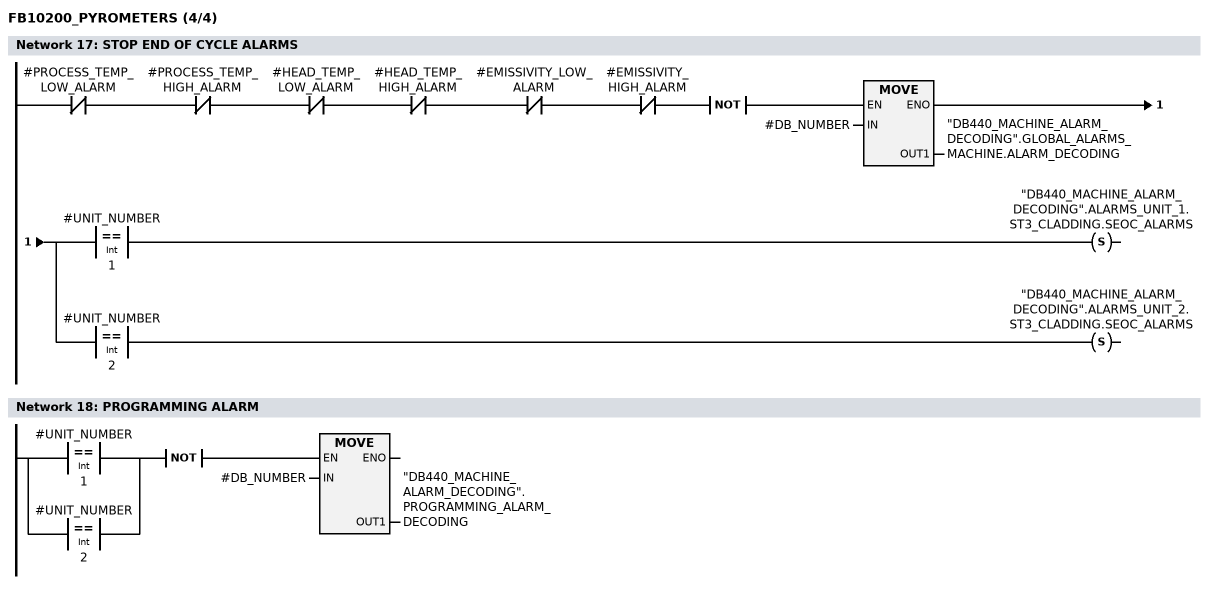
   RUNG wire#powerrail
      I_Contact( #PROCESS_TEMP_LOW_ALARM )
      I_Contact( #PROCESS_TEMP_HIGH_ALARM )
      I_Contact( #HEAD_TEMP_LOW_ALARM )
      I_Contact( #HEAD_TEMP_HIGH_ALARM )
      I_Contact( #EMISSIVITY_LOW_ALARM )
      I_Contact( #EMISSIVITY_HIGH_ALARM )
      Not()
      { S7_GenerateENO := "TRUE" } Move(in := #DB_NUMBER, out1 => "DB440_MACHINE_ALARM_DECODING".GLOBAL_ALARMS_MACHINE.ALARM_DECODING)
      wire#w1
      { S7_Templates := "SrcType := Int" } EQ_Contact(in1 := #UNIT_NUMBER, in2 := 1)
      S_Coil( "DB440_MACHINE_ALARM_DECODING".ALARMS_UNIT_1.ST3_CLADDING.SEOC_ALARMS )
   END_RUNG
   RUNG wire#w1
      { S7_Templates := "SrcType := Int" } EQ_Contact(in1 := #UNIT_NUMBER, in2 := 2)
      S_Coil( "DB440_MACHINE_ALARM_DECODING".ALARMS_UNIT_2.ST3_CLADDING.SEOC_ALARMS )
   END_RUNG
   // the same network as SCL:
   // ENO of a box is taken as its EN; it also drops when the box reports an error
   #_w1 := NOT (NOT #PROCESS_TEMP_LOW_ALARM AND NOT #PROCESS_TEMP_HIGH_ALARM AND NOT #HEAD_TEMP_LOW_ALARM AND NOT #HEAD_TEMP_HIGH_ALARM AND NOT #EMISSIVITY_LOW_ALARM AND NOT #EMISSIVITY_HIGH_ALARM);
   IF #_w1 THEN "DB440_MACHINE_ALARM_DECODING".GLOBAL_ALARMS_MACHINE.ALARM_DECODING := #DB_NUMBER; END_IF;
   IF #_w1 AND (#UNIT_NUMBER = 1) THEN
       "DB440_MACHINE_ALARM_DECODING".ALARMS_UNIT_1.ST3_CLADDING.SEOC_ALARMS := TRUE;
   END_IF;
   IF #_w1 AND (#UNIT_NUMBER = 2) THEN
       "DB440_MACHINE_ALARM_DECODING".ALARMS_UNIT_2.ST3_CLADDING.SEOC_ALARMS := TRUE;
   END_IF;
END_REGION

REGION Network 18: PROGRAMMING ALARM
   RUNG wire#powerrail
      { S7_Templates := "SrcType := Int" } EQ_Contact(in1 := #UNIT_NUMBER, in2 := 1)
      wire#w1
      Not()
      Move(in := #DB_NUMBER, out1 => "DB440_MACHINE_ALARM_DECODING".PROGRAMMING_ALARM_DECODING)
   END_RUNG
   RUNG wire#powerrail
      { S7_Templates := "SrcType := Int" } EQ_Contact(in1 := #UNIT_NUMBER, in2 := 2)
   END_RUNG wire#w1
   // the same network as SCL:
   IF NOT ((#UNIT_NUMBER = 1) OR (#UNIT_NUMBER = 2)) THEN
       "DB440_MACHINE_ALARM_DECODING".PROGRAMMING_ALARM_DECODING := #DB_NUMBER;
   END_IF;
END_REGION
END_FUNCTION_BLOCK
